// TIA Portal V20 export
DATA_BLOCK "AdjRight_DB"   // DB530
// stored: AutoNumber false, InstanceOfName AdjRight, InstanceOfType FB
"AdjRight"
   // VAR
   //    Var { ExternalAccessible := 'False'; ExternalVisible := 'False'; ExternalWritable := 'False'} : "TypeVar";
   //    Cmd { ExternalAccessible := 'False'; ExternalVisible := 'False'; ExternalWritable := 'False'} : "TypeCmd";
   //    Enc { ExternalAccessible := 'False'; ExternalVisible := 'False'; ExternalWritable := 'False'} : "SysCounterFast";
   //    Pos { ExternalAccessible := 'False'; ExternalVisible := 'False'; ExternalWritable := 'False'} : "SysPos";
   //    AdjSlow { ExternalAccessible := 'False'; ExternalVisible := 'False'; ExternalWritable := 'False'} : "SysMotor";
   //    AdjFast { ExternalAccessible := 'False'; ExternalVisible := 'False'; ExternalWritable := 'False'} : "SysLinMotC1150";
   //    TAutoOn { ExternalAccessible := 'False'; ExternalVisible := 'False'; ExternalWritable := 'False'} : TON_TIME;
   //    TAutoTarPosManOn { ExternalAccessible := 'False'; ExternalVisible := 'False'; ExternalWritable := 'False'} : TON_TIME;
   //    T { ExternalAccessible := 'False'; ExternalVisible := 'False'; ExternalWritable := 'False'} : Array[1..5] of IEC_TIMER;
   //    adjFastPnSlaveOff { ExternalAccessible := 'False'; ExternalVisible := 'False'; ExternalWritable := 'False'} : "SysPnSlaveDeactivate";
   //    tarOld { ExternalAccessible := 'False'; ExternalVisible := 'False'; ExternalWritable := 'False'} : DInt;
   //    autoTarPosMan { ExternalAccessible := 'False'; ExternalVisible := 'False'; ExternalWritable := 'False'} : Bool;
   //    setValueEnc { ExternalAccessible := 'False'; ExternalVisible := 'False'; ExternalWritable := 'False'} : Bool;
   //    autoRef { ExternalAccessible := 'False'; ExternalVisible := 'False'; ExternalWritable := 'False'} : Bool;
   //    posOld { ExternalAccessible := 'False'; ExternalVisible := 'False'; ExternalWritable := 'False'} : Real;
   //    posDiff { ExternalAccessible := 'False'; ExternalVisible := 'False'; ExternalWritable := 'False'} : Real;
   // END_VAR
BEGIN
END_DATA_BLOCK
